(* CODESYS project OOP example Interfaces using pointers or references.project

Project tree, tasks and I/O mapping:
  Device : CODESYS Control for Raspberry Pi SL, 3S - Smart Software Solutions GmbH, version 3.5.12.30
    application Application
      libraries: Standard, * (System); VisuDialogs, * (System); SysFile, 3.5.9.0 (System); AlarmManager, 3.5.12.0 (Intern)
      task MainTask (cyclic, interval 500 ms, priority 1, watchdog 1000 ms x 1) calls Interfaces_using_References, Interfaces_using_Pointers
      program Interfaces_using_References [ST]
      program Interfaces_using_Pointers [ST]
    SoftMotion General Axis Pool
    I²C
    SPI
    GPIOs_A_B : GPIOs B+/Pi2, 3S - Smart Software Solutions GmbH, version 3.5.11.0
        unmapped channels: digital inputs (GPIO0..GPIO31), digital outputs (GPIO0..GPIO31)
    Onewire
    Camera device
      <Empty>
  libraries: VisuSymbols, 3.5.10.0 (System)
  Interfaces/
    function block FB_Engine2 [ST]: MaxVelocity, Temperature, Velocity, Start, Stop
    interface ITF_Engine2: Start, Stop, MaxVelocity, Temperature, Velocity
    function block FB_NewEngine2 [ST]: Gear, Start
    interface ITF_NewEngine2: Gear
*)

// Device/Application/Interfaces_using_References
PROGRAM Interfaces_using_References
VAR
	fbEngine2   : FB_Engine2;
	fbNewEngine2: FB_NewEngine2;
	
	xWisselMotor: BOOL;
	RefMotor    : REFERENCE TO FB_Engine2;   // reference to Base class (a reference is a fixed pointer)

	rTemperature : REAL;
	xStart       : BOOL := TRUE;
	rMaxVelocity : REAL := 130; // kmph
	rVelocity    : REAL := 100; // kmph
	iGear : INT  := 1;
	xIsStarted   : BOOL;
	xStop        : BOOL; 
	
	I_NewEngine2: ITF_NewEngine2;   // instance of the the extended interface to test against via __QUERYINTERFACE( REFERENCE, ITF)
	iCurGear     : INT := 0;
	DoThis      : INT := 0;
	DoThat      : INT := 0;
END_VAR

// Switch the engine type to see the DoThis / DoThat counters 
IF NOT xWisselMotor THEN
   RefMotor REF= fbEngine2;
ELSE
   RefMotor REF= fbNewEngine2;
END_IF

IF xStart THEN
   xIsStarted := RefMotor.Start(rVelocity,iGear);    
	xStop 	    := FALSE;
ELSE        //alle anderen, motor uit
	xIsStarted := FALSE;
   xStop 		 := RefMotor.Stop(); 
END_IF

// AT runtime, the operator executes a TYPE conversion OF an INTERFACE REFERENCE into another TYPE. 
// The operator returns a BOOL result. TRUE means that CODESYS has performed the conversion successfully.
//
//__QUERYINTERFACE( <ITF_Source>, <ITF_Dest> );
//
// 1.Operand: Interface reference or FB interface
//
// 2.Operand: Interface reference with required target type
//
// The requirement for the explicit conversion is that both the ITF_Source and ITF_Dest are derived from Interface __System.IQueryInterface. 
// This interface is implicitly available does not require a library.

IF __QUERYINTERFACE( RefMotor, I_NewEngine2 ) THEN // perform the typecasting and test on conversion succes
   // DoThis++ dus FB_NewEngine2;
   DoThis := DoThis + 1;
   
   // read from the CASTED reference;
   iCurGear := I_NewEngine2.gear;
   
   // gear++
   iGear := iGear + 1;
   IF iCurGear >= 5 THEN 
      iGear := 1;                         
	END_IF
ELSE
   // DoThat++ FB_Engine2;
   DoThat := DoThat + 1;
END_IF;

RefMotor.MaxVelocity := rMaxVelocity;
rTemperature := RefMotor.Temperature;  

// toggle start;
xStart := NOT xStart;

END_PROGRAM

// Interfaces/FB_NewEngine2
FUNCTION_BLOCK FB_NewEngine2 EXTENDS FB_Engine2 IMPLEMENTS ITF_NewEngine2

// HAS GOT 2 METHODS;
// START has been redefined and a new Gear accessor has been added, just like in FB_NewEngine, only difference is the declaration via an Interface
SUPER^();

// new property to get / set the gear after start
PROPERTY Gear : INT
GET
Gear := THIS^._nGear;
END_GET
SET
THIS^._nGear := Gear;
END_SET
END_PROPERTY

METHOD Start : BOOL
VAR_INPUT
	fVelocity	: REAL;
	nGear	: INT;
END_VAR
// Overwriting an existing method (OVERRIDE)

// new: setting gear via property Gear setter
SUPER^.Start(nGear, TO_INT(fVelocity)); // calls Start() of FB_Engine, see below for explanation
Gear := nGear;


// SUPER^. POINTER
//In the above example, we created a new Start() METHOD in FB_NewEngine 
//and copied the existing code from FB_Engine into the new method. 
//This is not always possible, and it also runs counter to the principle of reuse!
//
//Consequently, every function block which is derived from another function block has access to a pointer called SUPER. 
//This can be used to access elements (methods, properties, local variables, etc.) from the parent function block.
//
//
//SUPER^.Start(nGear, fVelocity); // calls Start() of FB_Engine
//Gear := nGear;
//
//Instead of copying code from the parent function block to the new method, 
//the SUPER pointer can be used to call the method from the FB_Engine function block. 
//This does away with the need to copy the code.
END_METHOD

END_FUNCTION_BLOCK

// Interfaces/FB_Engine2
// An interface decouples methods and properties with re-usage in mind.
// The programmer now has the possibilty to write an interface once and use it in different function blocks
// 1) Define an interface like ITF_Engine_Interface and EXTEND this interface from __SYSTEM.IQUERYINTERFACE.
//       ^Extending the interface form iqueryInterface is *NOT* mandatory by default but it is very useful and thus should be *MANDATORY*!
// 2) Add methods and properties to the interface but do not write any code in them yet, just declare the "skeletton" 
// 3) to implement the interfaces on the FB itself, add the interface in the FB declaration: "IMPLEMENTS ITF_Engine_Interface"
// 4) right-click on the FB and select "Implement Interfaces", select a language (ST) and press ok the skeletons will be added to the tree of the FB
// 5) implement the sub code per method
// 6) End result is just like in FB_Engine, only difference is the declaration via an Interface!
FUNCTION_BLOCK FB_Engine2 IMPLEMENTS ITF_Engine2
VAR
   _xStarted   : BOOL;
   _fVelocity  : REAL;
   _MaxVelocity: REAL;
   _nGear      : INT;
   _Temperature: REAL;
END_VAR

PROPERTY MaxVelocity : REAL
GET
MaxVelocity := THIS^._MaxVelocity;
END_GET
SET
THIS^._MaxVelocity := MaxVelocity;
END_SET
END_PROPERTY

PROPERTY Temperature : REAL
GET
CASE TO_INT( THIS^._fVelocity ) OF // implicit typecasting(TO_INT), use REAL_TO_INT for explicit typecasting
   0..100 :
      THIS^._Temperature := 50;
   101..1000:
      THIS^._Temperature := 90;
   1001..10000:
      THIS^._Temperature := 100;
   10001..32767:
      THIS^._Temperature := 150;
END_CASE

Temperature := THIS^._Temperature;
END_GET
END_PROPERTY

PROPERTY Velocity : REAL
GET
Velocity := THIS^._fVelocity;
END_GET
END_PROPERTY

METHOD Start : BOOL
VAR_INPUT
	fVelocity	: REAL;
	nGear	: INT;
END_VAR
VAR
	rCurtemp : REAL;
END_VAR
THIS^._xStarted  := TRUE;
Start            := TRUE;
THIS^._nGear     := nGear;
THIS^._fVelocity := MIN( ABS( THIS^._MaxVelocity ), fVelocity );    // Beperk de nieuwe snelheid adhv de Maximum Snelheid
rCurtemp := THIS^.Temperature;
END_METHOD

METHOD Stop : BOOL
THIS^._xStarted := FALSE;
STOP            := TRUE;
END_METHOD

END_FUNCTION_BLOCK

// Interfaces/ITF_Engine2
// Note that the interface EXTENDS on the system basetype iQueryInterface. By this mechanisme we can "taste" wether this interface is correct for our purpose.
INTERFACE ITF_Engine2 EXTENDS __SYSTEM.IQueryInterface

METHOD Start : Bool;
VAR_INPUT
   fVelocity : REAL;
   nGear     : INT;
END_VAR
END_METHOD

METHOD Stop : BOOL
VAR_INPUT
END_VAR
END_METHOD

PROPERTY MaxVelocity : REAL
SET
END_SET
GET
END_GET
END_PROPERTY

PROPERTY Temperature : REAL
GET
END_GET
END_PROPERTY

PROPERTY Velocity : real
GET
END_GET
END_PROPERTY

END_INTERFACE

// Interfaces/ITF_NewEngine2
// Note that the interface EXTENDS on the ITF_NewEgine2, which in turn extended __System.iQueryInterface => make sure you understand this!
INTERFACE ITF_NewEngine2 EXTENDS ITF_Engine2

// new property to get / set the gear after start
PROPERTY Gear : int
SET
END_SET
GET
END_GET
END_PROPERTY

END_INTERFACE

// Device/Application/Interfaces_using_Pointers
PROGRAM Interfaces_using_Pointers
VAR
fbEngine2   : FB_Engine2;
fbNewEngine2: FB_NewEngine2;

xSwitchEngine: BOOL;
refEngine    : POINTER TO FB_Engine2;

rTemperature : REAL;
xStart       : BOOL := TRUE;
rMaxVelocity : REAL := 130; // kmph
rVelocity    : REAL := 100; // kmph
iGear : INT  := 1;
xIsStarted   : BOOL;
xStop        : BOOL; 

I_NewEngine2: ITF_NewEngine2;   // instance of the the extended interface to test against via __QUERYINTERFACE( REFERENCE, ITF)
iCurGear     : INT := 0;
iDoThis      : INT := 0;
iDoThat      : INT := 0;
END_VAR

// Switch the engine type to see the DoThis / DoThat counters 
IF NOT xSwitchEngine THEN
   refEngine := ADR(fbEngine2); // initialise pointer
ELSE
   refEngine := ADR(fbNewEngine2); // initialise pointer 
END_IF

IF xStart THEN
    xIsStarted := refEngine^.Start(rVelocity,iGear);       // both instances are called separatly
	xStop 	    := FALSE;
ELSE
    xIsStarted := FALSE;
   xStop 		 := refEngine^.Stop(); 
END_IF

// AT runtime, the operator executes a TYPE conversion OF an INTERFACE REFERENCE into another TYPE. 
// The operator returns a BOOL result. TRUE means that CODESYS has performed the conversion successfully.
//
//__QUERYINTERFACE( <ITF_Source>, <ITF_Dest> );
//
// 1.Operand: Interface reference or FB interface
//
// 2.Operand: Interface pointer with required target type
//
// The requirement for the explicit conversion is that both the ITF_Source and ITF_Dest are derived from Interface __System.IQueryInterface. 
// This interface is implicitly available does not require a library.

IF __QUERYINTERFACE( refEngine^, I_NewEngine2) THEN // perform the typecasting and test on conversion succes
   // DoThis++ dus FB_NewEngine2;
   iDoThis := iDoThis + 1;
   
   // read from the CASTED reference;
   iCurGear := I_NewEngine2.gear;
   
   // gear++
   iGear := iGear + 1;
   IF iCurGear >= 5 THEN 
      iGear := 1;                         
	END_IF
ELSE
   // DoThat++ dus FB_Engine2;
   iDoThat := iDoThat + 1;
END_IF;

refEngine^.MaxVelocity := rMaxVelocity;
rTemperature := refEngine^.Temperature;  

// toggle start;
xStart := NOT xStart;

END_PROGRAM
